{attribute 'qualified_only'}
VAR_GLOBAL
	arrDIs				 		AT %I*	: ARRAY[1..8] OF BOOL;
	arrDOs			 			AT %Q*	: ARRAY[1..4] OF BOOL;
	arrAIs						AT %I*	: ARRAY[1..2] OF INT;
	arrAOs						AT %Q*	: ARRAY[1..2] OF INT;
	leftAxis							: AXIS_REF;
	rightAxis							: AXIS_REF;
	
END_VAR

(* stored: Version 1.1.0.1
   GVL GVL_IO: Id {40eec583-8dde-47d2-ad44-37ec33bb6508} *)
